FUNCTION Convert_LWORD_TO_STRING : Hresult
VAR_INPUT
	in : LWORD;
	out : REFERENCE TO STRING;
END_VAR
VAR
	converted : STRING;
END_VAR

converted := LWORD_TO_STRING(in);

IF (STRING_TO_LWORD(converted) <> in) THEN
	Convert_LWORD_TO_STRING := INCOMPATIBLE;
	RETURN;
END_IF

out := converted;

END_FUNCTION

(* stored: Version 1.1.0.1, ProductVersion 3.1.4024.12
   POU Convert_LWORD_TO_STRING: Id {4eca8b6a-1c52-4f95-a4bf-f699d84555f7}, SpecialFunc None *)
